//{attribute 'qualified_only'}
VAR_GLOBAL
	iecCriticalSection : FB_IecCriticalSection; //must be used if communication routines are separated into their own core/task
END_VAR

(* stored: Version 1.1.0.1, ProductVersion 3.1.4024.11
   GVL Misc: Id {44a39edb-3d2a-49a6-af09-2a551348380e} *)
